DATA_BLOCK "DB_Cam_Output"
{ S7_Optimized_Access := 'FALSE' }
VERSION : 0.1
NON_RETAIN
   STRUCT
      Output : Array[0..127] of Byte;
   END_STRUCT;


BEGIN

END_DATA_BLOCK

